SUBAPPLICATION HW_2Sensors (* Subapplication Type *)
  (* Standard: 61499-2 *)
  (* Version 1.0, 2020-07-20, AK120569 *)
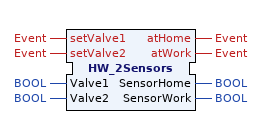
  EVENT_INPUT
    setValve1;
    setValve2;
  END_EVENT
  EVENT_OUTPUT
    atHome;
    atWork;
  END_EVENT
  VAR_INPUT
    Valve1 : BOOL;
    Valve2 : BOOL;
  END_VAR
  VAR_OUTPUT
    SensorHome : BOOL;
    SensorWork : BOOL;
  END_VAR
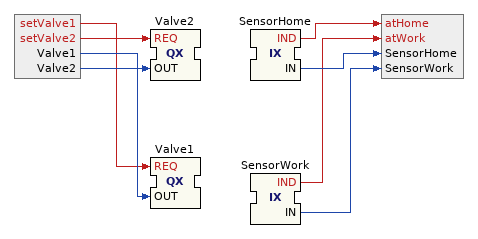
  FBS
    SensorWork : IX;
    Valve1 : QX;
    SensorHome : IX;
    Valve2 : QX;
  END_FBS
  EVENT_CONNECTIONS
    SensorHome.IND TO atHome;
    SensorWork.IND TO atWork;
    setValve2 TO Valve2.REQ;
    setValve1 TO Valve1.REQ;
  END_CONNECTIONS
  DATA_CONNECTIONS
    SensorHome.IN TO SensorHome;
    SensorWork.IN TO SensorWork;
    Valve1 TO Valve1.OUT;
    Valve2 TO Valve2.OUT;
  END_CONNECTIONS
END_SUBAPPLICATION
